// Mitsubishi GX Developer project: Traffic-Lights-GX-MItshubishi-PLC   PLC: FX2N

PROGRAM MAIN
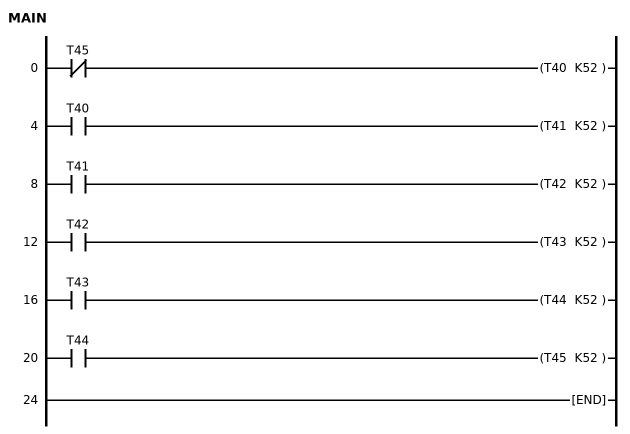
0     LDI     T45
      OUT     T40 K52
4     LD      T40
      OUT     T41 K52
8     LD      T41
      OUT     T42 K52
12    LD      T42
      OUT     T43 K52
16    LD      T43
      OUT     T44 K52
20    LD      T44
      OUT     T45 K52
24    END
END_PROGRAM
